# B&R Automation Studio project UaWrapper
Automation Studio 4.8.3.111 SP; Allows configuration of AR settings like IP address via an OPC UA method interface

## Configuration TestSetup

CPU X20CP1585, AutomationRuntime D4.63, Build 4.1.2, Vc V4.72.0

### Task classes (Cpu.sw)
```
Cyclic#4:
  UaCfg <- UaCfg.prg
Binaries: FWRules, TCData, udbdef, asfw, User, iomap, sysconf, arconfig, ashwd, Role, ashwac
Libraries: AsOpcUac, runtime, AsOpcUas, UasXTypes, asieccon, astime, AsARCfg, UasX, UasXARCfg
```

### Hardware
```
X20CP1585 : X20CP1585 v1.8.0.0
  Connector IF2:
    ActivateDevice = 1
  ConfigurationID = Config_TestSetup
  Simulation = 1
  ActivateOpcUa = 1
  OpcUaInformationModels_PV_Version = 1
```

## Logical view

Binary libraries used (declarations not repeated): operator, runtime, astime, AsIecCon, AsOpcUac, AsOpcUas, AsARCfg

### Package Logical/Libraries - Global libraries

### Library Logical/Libraries/UasX/UasXTypes (ANSIC) - OPC UA server functions
Depends on: AsOpcUac, AsOpcUas

#### Types.typ - Exported data types
```iecst
TYPE
	UasXMethodType : 	STRUCT
		fbOperate : UaSrv_MethodOperate;
		State : USINT;
		State_1 : USINT;
	END_STRUCT;
END_TYPE
```

#### Constants.var - Exported constants
```iecst
VAR CONSTANT
	UASX_ERR_NULL_POINTER : UINT := 50000;
END_VAR
```

#### UasXTypes.fun
```iecst
{REDUND_ERROR} FUNCTION _UasXDummy : BOOL (*dummy function to suppress warning 5880*) (*$GROUP=User,$CAT=User,$GROUPICON=User.png,$CATICON=User.png*)
END_FUNCTION
```

#### _UasXDummy.c
```c
#include <bur/plctypes.h>
#ifdef __cplusplus
	extern "C"
	{
#endif
	#include "UasXTypes.h"
#ifdef __cplusplus
	};
#endif
/* dummy function to suppress warning 5880 */
plcbit _UasXDummy(void)
{
	return 0;
}
```

### Library Logical/Libraries/UasX/UasX (ANSIC)
Depends on: AsOpcUas, UasXTypes

#### UasX.h
```c
#include <bur/plctypes.h>
#include <string.h>
#include <UasXTypes.h>

#define TRUE 1
#define FALSE 0

typedef UINT (*fpFubCallerType)(void* FubInstance);	// calls FUB and returns its status

/* macro to auto-generate fpFubCallerType function */
#define UASX_FUB_CALLER(FubType)\
static UINT FubType##Caller(void* FubInstance){\
	if (FubInstance == NULL) return UASX_ERR_NULL_POINTER;\
	struct FubType *fbInst = (struct FubType *)FubInstance;\
	FubType (fbInst);\
	return fbInst ->status;\
}

/* Cyclically process method object */
void UasXMethodOperate(struct UasXMethodType* Method, char* MethodName, fpFubCallerType fpFubCaller, void* FubInstance);
```

#### MethodOperate.c
```c
#include <UasX.h>

typedef enum {STATE_Init, STATE_CheckIsCalled, STATE_IsCalled, STATE_Finishing, STATE_Error = 255} StateEnum;
typedef enum {Good_Success = 0, Bad_InvalidState = 0x80AF0000} ErrorCodeEnum;

/* Cyclically process method object */
void UasXMethodOperate(struct UasXMethodType* Method, char* MethodName, fpFubCallerType fpFubCaller, void* FubInstance){
	if (MethodName == NULL) return;
	if (fpFubCaller == NULL) return;
	if (FubInstance == NULL) return;

	BOOL FirstCycleInState = (Method->State != Method->State_1);
	Method->State_1	= Method->State;

	switch (Method->State){
		case STATE_Init:
		case STATE_Error:
			Method->State	= STATE_CheckIsCalled;
			break;

		case STATE_CheckIsCalled:
			if (FirstCycleInState){
				Method->fbOperate.Execute	= FALSE;
				UaSrv_MethodOperate(&Method->fbOperate);
				strlcpy(Method->fbOperate.MethodName, MethodName, sizeof(Method->fbOperate.MethodName));
				Method->fbOperate.Execute	 = TRUE;
				Method->fbOperate.Action	 = UaMoa_CheckIsCalled;
			}
			UaSrv_MethodOperate(&Method->fbOperate);
			if (Method->fbOperate.Done){
				if (Method->fbOperate.IsCalled){
					Method->State	= STATE_IsCalled;
				}
				else {
					//remain in this state, call UaSrv_MethodOperate again
					Method->fbOperate.Execute	= FALSE;
					UaSrv_MethodOperate(&Method->fbOperate);
					Method->fbOperate.Execute	= TRUE;
				}
			}
			else if (Method->fbOperate.Error){
				Method->State	= STATE_Error;
			}
			break;

		case STATE_IsCalled:
			switch (fpFubCaller(FubInstance)){
				case ERR_FUB_BUSY:
					//do nothing, remain in state
					break;

				default:
					Method->State	= STATE_Finishing;
					break;
			}
			break;

		case STATE_Finishing:
			if (FirstCycleInState){
				Method->fbOperate.Execute	= FALSE;
				UaSrv_MethodOperate(&Method->fbOperate);
				Method->fbOperate.Execute	= TRUE;
				Method->fbOperate.Action	= UaMoa_Finished;
			}
			UaSrv_MethodOperate(&Method->fbOperate);
			if (Method->fbOperate.Done){
				Method->State	= STATE_CheckIsCalled;
			}
			else if (Method->fbOperate.Error){
				Method->State	= STATE_Error;
			}
			break;

		default:
			break;
	}
}
```

### Library Logical/Libraries/UasXARCfg (ANSIC)
Depends on: AsARCfg, UasXTypes

#### UasXARCfg.fun - Exported functions and function blocks
```iecst
{REDUND_ERROR} FUNCTION_BLOCK UasXCfgSetTimeZone (*OPC UA wrapper for CfgSetTimezone*) (*$GROUP=User,$CAT=User,$GROUPICON=User.png,$CATICON=User.png*)
	VAR_INPUT
		MethodName : STRING[255] := 'SetTimeZone'; (*Name of the method. *)
		TimezoneID : UINT; (*ID of the timezone you would like to set.*)
	END_VAR
	VAR_OUTPUT
		Status : UINT; (*Error number (0 = no error)*)
	END_VAR
	VAR
		Method : UasXMethodType;
		fbSetTimeZone : CfgSetTimeZone;
	END_VAR
END_FUNCTION_BLOCK

{REDUND_ERROR} FUNCTION_BLOCK UasXCfgSetIPAddr (*OPC UA wrapper for CfgSetIPAddr*) (*$GROUP=User,$CAT=User,$GROUPICON=User.png,$CATICON=User.png*)
	VAR_INPUT
		MethodName : STRING[255] := 'SetIPAddr'; (*Name of the method. *)
		Device : STRING[255] := 'IF2'; (*Device name (syntax: SL<x>.SS<y>.IF<z>)

Work with the following syntax when using a POWERLINK card:
V1		SL<x>.SS<y>.IF<z>.PLKETH
V2		SL<x>.SS<y>.IF<z>.ETH*)
		IPAddress : STRING[15]; (*IP address

Valid range "1.0.0.1" - "247.255.255.255"*)
	END_VAR
	VAR_OUTPUT
		Status : UINT; (*Error number (0 = no error)*)
	END_VAR
	VAR
		Method : UasXMethodType;
		fbSetIPAddr : CfgSetIPAddr;
	END_VAR
END_FUNCTION_BLOCK

{REDUND_ERROR} FUNCTION_BLOCK UasXCfgSetNtpClient (*OPC UA wrapper for CfgSetNtpClient*) (*$GROUP=User,$CAT=User,$GROUPICON=User.png,$CATICON=User.png*)
	VAR_INPUT
		MethodName : STRING[255] := 'SetNtpClient'; (*Name of the method. *)
		Start : BOOL; (*0: Stop client (cfgNTP_STOP)
1: Start client (cfgNTP_START)*)
		ServerAddress1 : STRING[15]; (*IP address of the 1st NTP server*)
		ServerAddress2 : STRING[15]; (*IP address of the 2nd NTP server*)
		ServerAddress3 : STRING[15]; (*IP address of the 3rd NTP server*)
		ServerAddress4 : STRING[15]; (*IP address of the 4th NTP server*)
	END_VAR
	VAR_OUTPUT
		Status : UINT; (*Error number (0 = no error)*)
	END_VAR
	VAR
		Method : UasXMethodType;
		fbSetNtpClient : CfgSetNtpClient;
	END_VAR
END_FUNCTION_BLOCK
```

#### UasXARCfg.c
```c
#include <bur/plctypes.h>
#include <UasX.h>
#ifdef __cplusplus
	extern "C"
	{
#endif
	#include "UasXARCfg.h"
#ifdef __cplusplus
	};
#endif

#define TRUE 1
#define FALSE 0

UASX_FUB_CALLER(CfgSetTimeZone);
UASX_FUB_CALLER(CfgSetIPAddr);
UASX_FUB_CALLER(CfgSetNtpClient);

/* OPC UA wrapper for CfgSetTimezone */
void UasXCfgSetTimeZone(struct UasXCfgSetTimeZone* inst)
{
	inst->fbSetTimeZone.enable		= TRUE;
	inst->fbSetTimeZone.option		= cfgOPTION_NON_VOLATILE;
	inst->fbSetTimeZone.timezoneID	= inst->TimezoneID;

	UasXMethodOperate(&inst->Method, inst->MethodName, CfgSetTimeZoneCaller, &inst->fbSetTimeZone);

	inst->Status	= inst->fbSetTimeZone.status;
}

/* OPC UA wrapper for CfgSetIPAddr */
void UasXCfgSetIPAddr(struct UasXCfgSetIPAddr* inst)
{
	inst->fbSetIPAddr.enable	= TRUE;
	inst->fbSetIPAddr.Option	= cfgOPTION_NON_VOLATILE;
	inst->fbSetIPAddr.pDevice	= (UDINT)inst->Device;
	inst->fbSetIPAddr.pIPAddr	= (UDINT)inst->IPAddress;

	UasXMethodOperate(&inst->Method, inst->MethodName, CfgSetIPAddrCaller, &inst->fbSetIPAddr);

	inst->Status	= inst->fbSetIPAddr.status;
}

/* OPC UA wrapper for CfgSetNtpClient */
void UasXCfgSetNtpClient(struct UasXCfgSetNtpClient* inst)
{
	inst->fbSetNtpClient.enable				= TRUE;
	inst->fbSetNtpClient.option				= cfgOPTION_NON_VOLATILE;
	inst->fbSetNtpClient.pServerAddress1	= (UDINT)inst->ServerAddress1;
	inst->fbSetNtpClient.pServerAddress2	= (UDINT)inst->ServerAddress2;
	inst->fbSetNtpClient.pServerAddress3	= (UDINT)inst->ServerAddress3;
	inst->fbSetNtpClient.pServerAddress4	= (UDINT)inst->ServerAddress4;
	inst->fbSetNtpClient.start				= inst->Start;

	UasXMethodOperate(&inst->Method, inst->MethodName, CfgSetNtpClientCaller, &inst->fbSetNtpClient);

	inst->Status	= inst->fbSetNtpClient.status;
}
```

### Program Logical/UaCfg (ANSIC)

#### Main.c - Init, cyclic, exit code
```c
#include <bur/plctypes.h>
#include "UasX.h"

#ifdef _DEFAULT_INCLUDES
#include <AsDefault.h>
#endif

void _INIT ProgramInit(void)
{
}

void _CYCLIC ProgramCyclic(void)
{
	UasXCfgSetTimeZone(&fbSetTimeZone);
	UasXCfgSetIPAddr(&fbSetIPAddr);
}

void _EXIT ProgramExit(void)
{
}
```

#### Variables.var - Local variables
```iecst
VAR
	fbSetTimeZone : UasXCfgSetTimeZone;
	fbSetIPAddr : UasXCfgSetIPAddr;
	fbSetNtpClient : UasXCfgSetNtpClient;
END_VAR
```

- Methods.uam (not shown)

Listed in the project but not available here: Logical/Global.typ, Logical/Global.var, Logical/Libraries/UasXARCfg/Types.typ, Logical/Libraries/UasXARCfg/Constants.var, Logical/UaCfg/Types.typ
